{attribute 'qualified_only'}
{attribute 'strict'}
TYPE DUT :
(
	Sick := 1,
	Pilz := 2,
	Parker :=3,
 	Bosch := 4
);
END_TYPE

(* stored: Version 1.1.0.1, ProductVersion 3.1.4024.12
   DUT DUT: Id {5192be19-3911-48b8-8692-ecab4bdd4558} *)
